ABB RAPID module: MainModule.mod

MODULE MainModule
LOCAL CONST string YuMi_App_Program_Version:="1.0.1"; !Do not edit or remove this line!
LOCAL VAR robtarget s43 := [[491.94,-308.73,64.10],[0.247601,0.742945,-0.619594,-0.0531904],[1,-3,0,1010],[118.165,9E+09,9E+09,9E+09,9E+09,9E+09]];
LOCAL VAR robtarget s42 := [[525.12,-108.90,15.96],[0.0331533,0.706346,-0.702887,-0.0769836],[1,-3,1,1010],[128.701,9E+09,9E+09,9E+09,9E+09,9E+09]];
LOCAL VAR robtarget s41 := [[453.36,-109.83,-4.37],[0.125812,0.720702,-0.668701,-0.132661],[1,-3,1,1010],[125.459,9E+09,9E+09,9E+09,9E+09,9E+09]];
LOCAL VAR robtarget s40 := [[461.61,-99.71,23.64],[0.133799,0.725083,-0.664379,-0.122283],[1,-3,1,1010],[132.237,9E+09,9E+09,9E+09,9E+09,9E+09]];
LOCAL VAR robtarget s39 := [[530.33,-200.43,75.47],[0.0798297,-0.859185,0.505215,-0.01362],[0,-3,0,1010],[148.999,9E+09,9E+09,9E+09,9E+09,9E+09]];
LOCAL VAR robtarget s38 := [[483.67,-298.42,39.41],[0.468265,-0.639664,0.502726,-0.344709],[0,-3,0,11],[149.982,9E+09,9E+09,9E+09,9E+09,9E+09]];
LOCAL VAR robtarget s37 := [[613.95,-232.75,83.31],[0.599586,-0.522262,0.444415,-0.412596],[1,-3,1,11],[137.21,9E+09,9E+09,9E+09,9E+09,9E+09]];
LOCAL VAR robtarget s36 := [[501.44,-102.97,10.11],[0.0823071,0.688996,-0.715276,-0.0830052],[1,-3,1,1010],[127.297,9E+09,9E+09,9E+09,9E+09,9E+09]];
LOCAL VAR robtarget s35 := [[453.76,-108.01,-5.22],[0.147909,0.699486,-0.689587,-0.115374],[1,-3,1,1010],[125.092,9E+09,9E+09,9E+09,9E+09,9E+09]];
LOCAL VAR robtarget s34 := [[456.75,-104.97,-0.82],[0.15612,0.706025,-0.684487,-0.0929117],[1,-3,1,1010],[126.243,9E+09,9E+09,9E+09,9E+09,9E+09]];
LOCAL VAR robtarget s33 := [[485.72,-106.64,73.18],[0.134057,0.68233,-0.706906,-0.129375],[1,-3,1,1010],[136.018,9E+09,9E+09,9E+09,9E+09,9E+09]];
LOCAL VAR robtarget s32 := [[414.31,-175.36,-14.67],[0.48775,-0.613567,0.508441,-0.356543],[0,-3,0,11],[164.194,9E+09,9E+09,9E+09,9E+09,9E+09]];
LOCAL VAR robtarget s31 := [[412.56,-183.06,-85.14],[0.428069,-0.649238,0.509798,-0.367902],[1,-3,0,11],[167.521,9E+09,9E+09,9E+09,9E+09,9E+09]];
LOCAL VAR robtarget s30 := [[415.46,-183.13,-80.05],[0.436643,-0.64254,0.502901,-0.378913],[1,-3,0,11],[167.779,9E+09,9E+09,9E+09,9E+09,9E+09]];
LOCAL VAR robtarget p1 := [[406.89,-179.86,-42.94],[0.329237,-0.738094,0.539563,-0.23599],[0,-3,0,11],[156.391,9E+09,9E+09,9E+09,9E+09,9E+09]];
LOCAL VAR robtarget s29 := [[388.28,-147.37,85.09],[0.177497,-0.0895413,0.838062,0.508064],[0,-2,0,1010],[144.786,9E+09,9E+09,9E+09,9E+09,9E+09]];
LOCAL VAR robtarget s28 := [[377.77,-240.64,-12.96],[0.0612554,0.396369,0.864911,0.301776],[0,-2,1,1010],[135.784,9E+09,9E+09,9E+09,9E+09,9E+09]];
LOCAL VAR robtarget s27 := [[377.77,-240.64,-12.96],[0.0612635,0.396357,0.864909,0.301795],[0,-2,1,1010],[135.784,9E+09,9E+09,9E+09,9E+09,9E+09]];
LOCAL VAR robtarget s26 := [[375.45,-120.15,9.01],[0.29088,0.594444,0.599765,0.449786],[1,-1,0,1010],[138.471,9E+09,9E+09,9E+09,9E+09,9E+09]];
LOCAL VAR robtarget s25 := [[433.47,-113.73,-15.91],[0.346506,0.584015,0.590385,0.436241],[1,-1,0,1010],[138.938,9E+09,9E+09,9E+09,9E+09,9E+09]];
LOCAL VAR robtarget s24 := [[430.73,-112.58,-2.80],[0.352418,0.570416,0.590717,0.448866],[1,-1,0,1010],[138.366,9E+09,9E+09,9E+09,9E+09,9E+09]];
LOCAL VAR robtarget s23 := [[448.55,-124.34,51.61],[0.22769,0.533492,0.668437,0.465549],[1,-1,0,1010],[131.291,9E+09,9E+09,9E+09,9E+09,9E+09]];
LOCAL VAR robtarget s22 := [[474.01,-193.16,22.86],[0.134201,-0.611281,-0.76704,0.14133],[1,-1,1,11],[139.503,9E+09,9E+09,9E+09,9E+09,9E+09]];
LOCAL VAR robtarget s21 := [[428.62,-176.27,-83.17],[0.138692,-0.615453,-0.765706,0.125207],[1,-1,1,11],[149.965,9E+09,9E+09,9E+09,9E+09,9E+09]];
LOCAL VAR robtarget s20 := [[455.96,-175.33,67.49],[0.425487,0.51878,0.587505,0.452399],[0,-3,-2,11],[-177.346,9E+09,9E+09,9E+09,9E+09,9E+09]];
LOCAL VAR robtarget s19 := [[411.66,-192.15,16.54],[0.181981,0.62416,0.722418,0.235415],[0,-3,2,11],[172.986,9E+09,9E+09,9E+09,9E+09,9E+09]];
LOCAL VAR robtarget s18 := [[425.56,-179.34,-78.05],[0.160724,0.587013,0.768308,0.198205],[0,-3,2,11],[166.895,9E+09,9E+09,9E+09,9E+09,9E+09]];
LOCAL VAR robtarget s17 := [[410.33,-174.58,-17.85],[0.145859,0.613451,0.762207,0.146437],[0,-2,2,11],[157.417,9E+09,9E+09,9E+09,9E+09,9E+09]];
LOCAL VAR robtarget s16 := [[432.43,-181.71,-47.22],[0.179519,-0.636686,-0.735627,0.145799],[1,-1,1,11],[156.736,9E+09,9E+09,9E+09,9E+09,9E+09]];
LOCAL VAR robtarget s15 := [[508.88,-162.80,16.30],[0.0119494,-0.682961,-0.728524,0.0517069],[1,-2,1,11],[164.288,9E+09,9E+09,9E+09,9E+09,9E+09]];
LOCAL VAR robtarget s14 := [[557.16,-113.79,46.21],[0.0312457,0.71325,0.696451,0.0724836],[1,-2,1,11],[-156.654,9E+09,9E+09,9E+09,9E+09,9E+09]];
LOCAL VAR robtarget s13 := [[469.10,-114.11,-53.63],[0.00905563,-0.696852,-0.716973,0.0162871],[1,-2,1,11],[-162.459,9E+09,9E+09,9E+09,9E+09,9E+09]];
LOCAL VAR robtarget s12 := [[474.67,-114.46,-39.47],[0.01248,-0.700622,-0.712864,0.0282491],[1,-2,1,11],[-160.647,9E+09,9E+09,9E+09,9E+09,9E+09]];
LOCAL VAR robtarget s11 := [[473.23,-126.88,63.00],[0.0237144,0.658653,0.739848,0.135049],[0,-2,1,11],[-145.561,9E+09,9E+09,9E+09,9E+09,9E+09]];
LOCAL VAR robtarget s10 := [[381.69,-96.96,17.16],[0.13894,0.402231,0.839987,0.336643],[0,-2,0,11],[-119.721,9E+09,9E+09,9E+09,9E+09,9E+09]];
LOCAL VAR robtarget s9 := [[390.33,-74.42,-67.11],[0.125269,0.387862,0.876169,0.257292],[1,-2,0,11],[-117.738,9E+09,9E+09,9E+09,9E+09,9E+09]];
LOCAL VAR robtarget s8 := [[469.53,-113.48,-54.32],[0.00884111,-0.689554,-0.723758,0.0247353],[1,-2,1,11],[-157.568,9E+09,9E+09,9E+09,9E+09,9E+09]];
LOCAL VAR robtarget s7 := [[474.18,-111.46,-49.11],[0.0245295,0.684802,0.727037,-0.0431526],[1,-2,1,11],[-157.233,9E+09,9E+09,9E+09,9E+09,9E+09]];
LOCAL VAR robtarget s6 := [[479.64,-138.68,31.69],[0.00246183,-0.670817,-0.741,0.0302848],[1,-2,1,11],[-130.321,9E+09,9E+09,9E+09,9E+09,9E+09]];
LOCAL VAR robtarget s5 := [[385.22,-154.60,12.05],[0.127122,0.413938,0.865263,0.252616],[0,-2,0,11],[-116.902,9E+09,9E+09,9E+09,9E+09,9E+09]];
LOCAL VAR robtarget s4 := [[390.36,-74.56,-67.12],[0.125372,0.387879,0.876179,0.257181],[1,-2,0,11],[-117.733,9E+09,9E+09,9E+09,9E+09,9E+09]];
LOCAL VAR robtarget s3 := [[385.07,-81.86,-65.27],[0.137555,0.41703,0.865727,0.24017],[1,-2,0,11],[-112.918,9E+09,9E+09,9E+09,9E+09,9E+09]];
LOCAL VAR robtarget s2 := [[364.79,-83.02,-15.45],[0.136492,0.363321,0.891617,0.23321],[0,-2,0,11],[-115.842,9E+09,9E+09,9E+09,9E+09,9E+09]];
LOCAL VAR robtarget s1 := [[358.40,-68.21,133.32],[0.275578,0.0423399,0.862981,0.42134],[0,-2,-1,11],[-117.323,9E+09,9E+09,9E+09,9E+09,9E+09]];
PROC main()
MoveSync s1;
MoveSync s2;
MoveSync s3;
MoveSync s9;
CloseHand;
MoveSync s10;
MoveSync s11;
MoveSync s12;
MoveSync s13;
OpenHand;
MoveSync s14;
MoveSync s15;
MoveSync s17;
Move p1;
MoveSync s30;
MoveSync s31;
CloseHand;
MoveSync s32;
MoveSync s38;
MoveSync s39;
MoveSync s40;
MoveSync s41;
OpenHand;
MoveSync s42;
MoveSync s43;
ENDPROC
ENDMODULE
